// TIA Portal V16 export
// export: Created 2024-12-03T15:41:45.6527845Z, ExportSetting WithReadOnly, DisplayName Totally Integrated Automation Portal, DisplayVersion V16 Update 6, DisplayName TIA Portal Version Control Interface, DisplayVersion V16 Update 2, DisplayName TIA Portal Openness, DisplayVersion V16 Update 6, DisplayName TIA Portal Teamcenter Gateway, DisplayVersion V16, DisplayName SINAMICS Startdrive Advanced, DisplayVersion V16 Update 5, DisplayName SINAMICS Startdrive G130, G150, S120, S150, SINAMICS MV, S210, DisplayVersion V16 Update 5, DisplayName SINAMICS Startdrive G110M, G120, G120C, G120D, G120P, G115D, DisplayVersion V16 Update 5, DisplayName STEP 7 Professional, DisplayVersion V16 Update 6, DisplayName STEP 7 Safety, DisplayVersion V16, DisplayName WinCC Advanced / Unified PC, DisplayVersion V16 Update 6
TYPE "SKU_In_Data_UDT"
// stored: CreationDate 2023-04-19T11:30:38.0051651Z, InterfaceModifiedDate 2023-04-19T12:03:36.1474172Z, IsConsistent true, LibraryConformanceStatus The object is library-conformant., ModifiedDate 2023-04-19T12:03:36.1474172Z
   STRUCT
      reserve7 : Byte;
      Input_1 : Bool;
      Input_2 : Bool;
      reserve1 : Bool;
      reserve2 : Bool;
      reserve3 : Bool;
      reserve4 : Bool;
      reserve5 : Bool;
      reserve6 : Bool;
   END_STRUCT;
END_TYPE
